FUNCTION_BLOCK EQ_Piston (* Piston, DC motor through an L298N (IN3 up, IN4 down, ENB speed) with a limit switch at the working position; equipment IO: owns its IO points; commands Stop=0, Up=1, Down=2 *)
  (* Standard: 61499-2 *)
  (* Version 0.1, 2026-09-28, Project contributors, AAU Smart Production Lab *)
  PACKAGE stoppering;
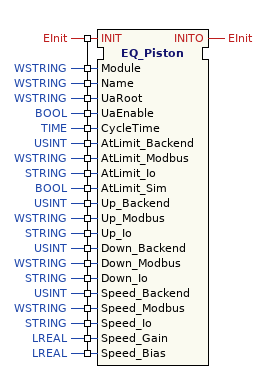
  EVENT_INPUT
    INIT : EInit WITH Module, Name, UaRoot, UaEnable, CycleTime, AtLimit_Backend, AtLimit_Modbus, AtLimit_Io, AtLimit_Sim, Up_Backend, Up_Modbus, Up_Io, Down_Backend, Down_Modbus, Down_Io, Speed_Backend, Speed_Modbus, Speed_Io, Speed_Gain, Speed_Bias;
  END_EVENT
  EVENT_OUTPUT
    INITO : EInit;
  END_EVENT
  VAR_INPUT
    Module : WSTRING;
    Name : WSTRING := "Piston";
    UaRoot : WSTRING;
    UaEnable : BOOL;
    CycleTime : TIME := T#50ms;
    AtLimit_Backend : USINT := 2;
    AtLimit_Modbus : WSTRING;
    AtLimit_Io : STRING;
    AtLimit_Sim : BOOL := FALSE;
    Up_Backend : USINT := 2;
    Up_Modbus : WSTRING;
    Up_Io : STRING;
    Down_Backend : USINT := 2;
    Down_Modbus : WSTRING;
    Down_Io : STRING;
    Speed_Backend : USINT := 2;
    Speed_Modbus : WSTRING;
    Speed_Io : STRING;
    Speed_Gain : LREAL := 257.0;
    Speed_Bias : LREAL := 0.0;
  END_VAR
  FBS
    Logic : stoppering::EL_Piston;
    Mode : modlib::MOD_StateView;
    SubCmd : iec61499::net::SUBSCRIBE_4(QI := TRUE);
    PubState : iec61499::net::PUBLISH_2(QI := TRUE);
    PubUa : iec61499::net::PUBLISH_1;
    In_AtLimit : modlib::IO_DI;
    Out_Up : modlib::IO_DO;
    Out_Down : modlib::IO_DO;
    Out_Speed : modlib::IO_AO;
    Cycle : iec61499::events::E_CYCLE;
    PhaseT : iec61499::events::E_DELAY;
  END_FBS
  EVENT_CONNECTIONS
    INIT TO Logic.INIT;
    Logic.INITO TO Mode.INIT;
    Mode.INITO TO SubCmd.INIT;
    SubCmd.INITO TO PubState.INIT;
    PubState.INITO TO PubUa.INIT;
    PubUa.INITO TO In_AtLimit.INIT;
    In_AtLimit.INITO TO Out_Up.INIT;
    Out_Up.INITO TO Out_Down.INIT;
    Out_Down.INITO TO Out_Speed.INIT;
    Out_Speed.INITO TO Cycle.START;
    Out_Speed.INITO TO INITO;
    SubCmd.IND TO Logic.CMD;
    Mode.CHG TO Logic.MOD_CHG;
    Cycle.EO TO Logic.REFRESH;
    Cycle.EO TO In_AtLimit.REQ;
    In_AtLimit.CNF TO Logic.SAMPLE;
    Logic.STATE TO PubState.REQ;
    Logic.STATE TO PubUa.REQ;
    Logic.DRIVE TO Out_Up.REQ;
    Out_Up.CNF TO Out_Down.REQ;
    Out_Down.CNF TO Out_Speed.REQ;
    Out_Speed.CNF TO Logic.DRIVEN;
    Logic.PHASE_START TO PhaseT.START;
    Logic.PHASE_STOP TO PhaseT.STOP;
    PhaseT.EO TO Logic.PHASE_T;
  END_CONNECTIONS
  DATA_CONNECTIONS
    Module TO Logic.Module;
    Name TO Logic.Name;
    UaRoot TO Logic.UaRoot;
    Module TO Mode.Module;
    Logic.IdCmd TO SubCmd.ID;
    Logic.IdState TO PubState.ID;
    Logic.IdPub TO PubUa.ID;
    UaEnable TO PubUa.QI;
    CycleTime TO Cycle.DT;
    SubCmd.RD_1 TO Logic.C_Holder;
    SubCmd.RD_2 TO Logic.C_Command;
    SubCmd.RD_3 TO Logic.C_Arg;
    SubCmd.RD_4 TO Logic.C_Release;
    Mode.State TO Logic.ModState;
    AtLimit_Backend TO In_AtLimit.Backend;
    AtLimit_Modbus TO In_AtLimit.ModbusId;
    AtLimit_Io TO In_AtLimit.IoName;
    AtLimit_Sim TO In_AtLimit.SimValue;
    In_AtLimit.IN TO Logic.I_AtLimit;
    Logic.AtLimit TO PubState.SD_1;
    Logic.AtLimit TO PubUa.SD_1;
    Logic.Holder TO PubState.SD_2;
    Up_Backend TO Out_Up.Backend;
    Up_Modbus TO Out_Up.ModbusId;
    Up_Io TO Out_Up.IoName;
    Logic.O_Up TO Out_Up.OUT;
    Down_Backend TO Out_Down.Backend;
    Down_Modbus TO Out_Down.ModbusId;
    Down_Io TO Out_Down.IoName;
    Logic.O_Down TO Out_Down.OUT;
    Speed_Backend TO Out_Speed.Backend;
    Speed_Modbus TO Out_Speed.ModbusId;
    Speed_Io TO Out_Speed.IoName;
    Logic.O_Speed TO Out_Speed.OUT;
    Logic.E_Speed TO Out_Speed.EN;
    Speed_Gain TO Out_Speed.Gain;
    Speed_Bias TO Out_Speed.Bias;
    Logic.PhaseDT TO PhaseT.DT;
  END_CONNECTIONS
END_FUNCTION_BLOCK
